IF (EipIntInput[7]=1 AND nOldEipInput[7]<>1) OR exeStop_os THEN
	exeStop_os := FALSE;
	exeStop := NOT exeStop;
	EipIntOutput[8] := 1 - EipIntOutput[8];
END_IF
nOldEipInput[7] := EipIntInput[7];

IF EipIntInput[8]=1 OR exeresetPB THEN
	exeresetPB := FALSE;
	exereset := TRUE;
//ELSE
//	exereset := FALSE;
END_IF

IF EipIntInput[9]=1 OR exerestartPB THEN
	exerestart := TRUE;
ELSE
	exerestart := FALSE;
END_IF

FOR i:=1 TO 2 DO
	IF bMoverEnable[i]= TRUE THEN
		EipIntOutput[i] :=1;
	ELSE
		EipIntOutput[i] :=0;
	END_IF
	IF bMoverDisable[i]= TRUE THEN
		EipIntOutput[i+2] :=1;
	ELSE
		EipIntOutput[i+2] :=0;
	END_IF
END_FOR

//速度変数を外部PLCから変更
IF EipIntInput[10] <> nOldEipInput[10] THEN
	ValueV := EipIntInput[10];
	nOldEipInput[10] := EipIntInput[10];
END_IF
EipIntOutput[6] := ValueV;
IF EipIntInput[11] <> nOldEipInput[11] THEN
	ValueC := EipIntInput[11];
	nOldEipInput[11] := EipIntInput[11];
END_IF
EipIntOutput[7] := ValueC;

IF fbAutoScan.bDone THEN
	EipIntOutput[9] := 1;
ELSE
	EipIntOutput[9] := 0;
END_IF
END_ACTION

END_PROGRAM

// ---- POUs/FB/FB_XpEnableMover.TcPOU
FUNCTION_BLOCK FB_XpEnableMover
VAR_IN_OUT
	XpMover							: MC_PlanarMover;
	XpGroup							: MC_PlanarGroup;
END_VAR
VAR_INPUT
	execute							: BOOL;
END_VAR
VAR_OUTPUT
	done							: BOOL;
	busy							: BOOL;
	error							: BOOL;
	aborted							: BOOL;
END_VAR
VAR
	_XpFeedback						: ARRAY [0.._MAX_XPLANAR_FEEDBACK] OF MC_PlanarFeedback;
END_VAR
VAR
	_sequence						: UINT;
	_i								: UINT;
	_countError						: UINT;
END_VAR
VAR CONSTANT
	_MAX_XPLANAR_FEEDBACK			: UINT := 1;
	_MAX_COUNT_ERROR				: UINT := 5;
	
	_INIT							: UINT := 0000;
	_READY							: UINT := 0001;
	_ENABLE_MOVER					: UINT := 0011;
	_CHECK_ENABLE_MOVER				: UINT := 0012;
	_ADD_TO_GROUP					: UINT := 0013;
	_CHECK_ADD_TO_GROUP				: UINT := 0014;
	_DONE							: UINT := 1000;
	_ERROR							: UINT := 2000;
	_ABORTED						: UINT := 3000;
END_VAR

updateXPlanarFB();
CASE _sequence OF
	_INIT:
		_sequence := _READY;	

	_READY:
		IF execute THEN
			busy := TRUE;
			_sequence := _ENABLE_MOVER;
		END_IF

	_ENABLE_MOVER:
		XpMover.Enable(commandFeedback:= _XpFeedback[0]);
		_sequence := _CHECK_ENABLE_MOVER;
	
	_CHECK_ENABLE_MOVER:
		IF _XpFeedback[0].Done THEN
			_countError := 0;
			_sequence := _ADD_TO_GROUP;
		ELSIF _XpFeedback[0].Error THEN
			_countError := _countError + 1;
			_sequence := _ENABLE_MOVER;
		END_IF
		IF _countError > _MAX_COUNT_ERROR THEN
			_countError := 0;
			_sequence := _ERROR;
		END_IF
	
	_ADD_TO_GROUP:
		XpMover.AddToGroup(commandFeedback:= _XpFeedback[1], group:= XpGroup);
		_sequence := _CHECK_ADD_TO_GROUP;
	
	_CHECK_ADD_TO_GROUP:
		IF _XpFeedback[1].Done THEN
			_countError := 0;
			_sequence := _DONE;
		ELSIF _XpFeedback[1].Error THEN
			_countError := _countError + 1;
			_sequence := _ADD_TO_GROUP;
		END_IF
		IF _countError > _MAX_COUNT_ERROR THEN
			_countError := 0;
			_sequence := _ERROR;
		END_IF
	
	_DONE:
		done := TRUE;
		busy := FALSE;
		IF NOT execute THEN
			done := FALSE;
			_sequence := _READY;
		END_IF
		
	_ERROR:
		error := TRUE;
		busy := FALSE;
		IF NOT execute THEN
			error := FALSE;
			_sequence := _READY;
		END_IF
		
	_ABORTED:
		aborted := TRUE;
		busy := FALSE;
		IF NOT execute THEN
			aborted := FALSE;
			_sequence := _READY;
		END_IF
END_CASE

ACTION updateXPlanarFB:
FOR _i:=0 TO _MAX_XPLANAR_FEEDBACK DO
	_XpFeedback[_i].Update();
END_FOR
END_ACTION

END_FUNCTION_BLOCK

// ---- POUs/FB/FB_XpDisableMover.TcPOU
FUNCTION_BLOCK FB_XpDisableMover
VAR_IN_OUT
	XpMover							: MC_PlanarMover;
	XpGroup							: MC_PlanarGroup;
END_VAR
VAR_INPUT
	execute							: BOOL;
END_VAR
VAR_OUTPUT
	done							: BOOL;
	busy							: BOOL;
	error							: BOOL;
	aborted							: BOOL;
END_VAR
VAR
	_XpFeedback						: ARRAY [0.._MAX_XPLANAR_FEEDBACK] OF MC_PlanarFeedback;
END_VAR
VAR
	_sequence						: UINT;
	_i								: UINT;
	_countError						: UINT;
END_VAR
VAR CONSTANT
	_MAX_XPLANAR_FEEDBACK			: UINT := 1;
	_MAX_COUNT_ERROR				: UINT := 5;
	
	_INIT							: UINT := 0000;
	_READY							: UINT := 0001;
	_REMOVE_FROM_GROUP				: UINT := 0011;
	_CHECK_REMOVE_FROM_GROUP		: UINT := 0012;
	_DISABLE_MOVER					: UINT := 0013;
	_CHECK_DISABLE_MOVER			: UINT := 0014;
	_DONE							: UINT := 1000;
	_ERROR							: UINT := 2000;
	_ABORTED						: UINT := 3000;
END_VAR

updateXPlanarFB();
CASE _sequence OF
	_INIT:
		_sequence := _READY;
		
	_READY:
		IF execute THEN
			busy := TRUE;
			_sequence := _REMOVE_FROM_GROUP;
		END_IF

	_REMOVE_FROM_GROUP:
		XpMover.RemoveFromGroup(commandFeedback:= _XpFeedback[0]);
		_sequence := _CHECK_REMOVE_FROM_GROUP;
	
	_CHECK_REMOVE_FROM_GROUP:
		IF _XpFeedback[0].Done THEN
			_countError := 0;
			_sequence := _DISABLE_MOVER;
		ELSIF _XpFeedback[0].Error THEN
			_countError := _countError + 1;
			_sequence := _REMOVE_FROM_GROUP;
		END_IF
		IF _countError > _MAX_COUNT_ERROR THEN
			_countError := 0;
			_sequence := _ERROR;
		END_IF
	
	_DISABLE_MOVER:
		XpMover.Disable(commandFeedback:= _XpFeedback[1]);
		_sequence := _CHECK_DISABLE_MOVER;
	
	_CHECK_DISABLE_MOVER:
		IF _XpFeedback[1].Done THEN
			_countError := 0;
			_sequence := _DONE;
		ELSIF _XpFeedback[1].Error THEN
			_countError := _countError + 1;
			_sequence := _DISABLE_MOVER;
		END_IF
		IF _countError > _MAX_COUNT_ERROR THEN
			_countError := 0;
			_sequence := _ERROR;
		END_IF
	
	_DONE:
		done := TRUE;
		busy := FALSE;
		IF NOT execute THEN
			done := FALSE;
			_sequence := _READY;
		END_IF
		
	_ERROR:
		error := TRUE;
		busy := FALSE;
		IF NOT execute THEN
			error := FALSE;
			_sequence := _READY;
		END_IF
		
	_ABORTED:
		aborted := TRUE;
		busy := FALSE;
		IF NOT execute THEN
			aborted := FALSE;
			_sequence := _READY;
		END_IF
END_CASE

ACTION updateXPlanarFB:
FOR _i:=0 TO _MAX_XPLANAR_FEEDBACK DO
	_XpFeedback[_i].Update();
END_FOR
END_ACTION

END_FUNCTION_BLOCK

// ---- POUs/FB/FB_XpEnableGroup.TcPOU
FUNCTION_BLOCK FB_XpEnableGroup
VAR_IN_OUT
	XpGroup							: MC_PlanarGroup;
END_VAR
VAR_INPUT
	execute							: BOOL;
END_VAR
VAR_OUTPUT
	done							: BOOL;
	busy							: BOOL;
	error							: BOOL;
	aborted							: BOOL;
END_VAR
VAR
	_XpFeedback						: ARRAY [0.._MAX_XPLANAR_FEEDBACK] OF MC_PlanarFeedback;
END_VAR
VAR
	_sequence						: UINT;
	_i								: UINT;
	_countError						: UINT;
END_VAR
VAR CONSTANT
	_MAX_XPLANAR_FEEDBACK			: UINT := 1;
	_MAX_COUNT_ERROR				: UINT := 5;
	
	_INIT							: UINT := 0000;
	_READY							: UINT := 0001;
	_ENABLE_GROUP					: UINT := 0011;
	_CHECK_ENABLE_GROUP				: UINT := 0012;
	_DONE							: UINT := 1000;
	_ERROR							: UINT := 2000;
	_ABORTED						: UINT := 3000;
END_VAR

updateXPlanarFB();
CASE _sequence OF
	_INIT:
		_sequence := _READY;
		
	_READY:
		IF execute THEN
			busy := TRUE;
			_sequence := _ENABLE_GROUP;
		END_IF

	_ENABLE_GROUP:
		XpGroup.Enable(commandFeedback:= _XpFeedback[0]);
		_sequence := _CHECK_ENABLE_GROUP;
	
	_CHECK_ENABLE_GROUP:
		IF _XpFeedback[0].Done THEN
			_countError := 0;
			_sequence := _DONE;
		ELSIF _XpFeedback[0].Error THEN
			_countError := _countError + 1;
			_sequence := _ENABLE_GROUP;
		END_IF
		IF _countError > _MAX_COUNT_ERROR THEN
			_countError := 0;
			_sequence := _ERROR;
		END_IF
	_DONE:
		done := TRUE;
		busy := FALSE;
		IF NOT execute THEN
			done := FALSE;
			_sequence := _READY;
		END_IF
		
	_ERROR:
		error := TRUE;
		busy := FALSE;
		IF NOT execute THEN
			error := FALSE;
			_sequence := _READY;
		END_IF
		
	_ABORTED:
		aborted := TRUE;
		busy := FALSE;
		IF NOT execute THEN
			aborted := FALSE;
			_sequence := _READY;
		END_IF
END_CASE

ACTION updateXPlanarFB:
FOR _i:=0 TO _MAX_XPLANAR_FEEDBACK DO
	_XpFeedback[_i].Update();
END_FOR
END_ACTION

END_FUNCTION_BLOCK

// ---- POUs/FB/FB_XpEnableEnvironment.TcPOU
FUNCTION_BLOCK FB_XpEnableEnvironment
VAR_IN_OUT
	XpEnvironment					: MC_PlanarEnvironment;
	XpGroup							: MC_PlanarGroup;
END_VAR
VAR_INPUT
	execute							: BOOL;
END_VAR
VAR_OUTPUT
	done							: BOOL;
	busy							: BOOL;
	error							: BOOL;
	aborted							: BOOL;
END_VAR
VAR
	_XpFeedback						: ARRAY [0.._MAX_XPLANAR_FEEDBACK] OF MC_PlanarFeedback;
END_VAR
VAR
	_sequence						: UINT;
	_i								: UINT;
	_countError						: UINT;
END_VAR
VAR CONSTANT
	_MAX_XPLANAR_FEEDBACK			: UINT := 1;
	_MAX_COUNT_ERROR				: UINT := 5;
	
	_INIT							: UINT := 0000;
	_READY							: UINT := 0001;
	_CREATE_BOUNDARY				: UINT := 0011;
	_CHECK_CREATE_BOUNDARY			: UINT := 0012;
	_ENVIRONMENT_ADD_TO_GROUP		: UINT := 0013;
	_CHECK_ENVIRONMENT_ADD_TO_GROUP	: UINT := 0014;
	_DONE							: UINT := 1000;
	_ERROR							: UINT := 2000;
	_ABORTED						: UINT := 3000;
END_VAR

updateXPlanarFB();
CASE _sequence OF
	_INIT:
		_sequence := _READY;
		
	_READY:
		IF execute THEN
			busy := TRUE;
			_sequence := _CREATE_BOUNDARY;
		END_IF
		
	_CREATE_BOUNDARY:
		XpEnvironment.CreateBoundary(commandFeedback:= _XpFeedback[0]);
		_sequence := _CHECK_CREATE_BOUNDARY;
	
	_CHECK_CREATE_BOUNDARY:
		IF _XpFeedback[0].Done THEN
			_countError := 0;
			_sequence := _ENVIRONMENT_ADD_TO_GROUP;
		ELSIF _XpFeedback[0].Error THEN
			_countError := _countError + 1;
			_sequence := _CREATE_BOUNDARY;
		END_IF
		IF _countError > _MAX_COUNT_ERROR THEN
			_countError := 0;
			_sequence := _ERROR;
		END_IF
	
	_ENVIRONMENT_ADD_TO_GROUP:
		XpEnvironment.AddToGroup(commandFeedback:= _XpFeedback[1], group:= XpGroup);
		_sequence := _CHECK_ENVIRONMENT_ADD_TO_GROUP;
	
	_CHECK_ENVIRONMENT_ADD_TO_GROUP:
		IF _XpFeedback[1].Done THEN
			_countError := 0;
			_sequence := _DONE;
		ELSIF _XpFeedback[1].Error THEN
			_countError := _countError + 1;
			_sequence := _ENVIRONMENT_ADD_TO_GROUP;
		END_IF
		IF _countError > _MAX_COUNT_ERROR THEN
			_countError := 0;
			_sequence := _ERROR;
		END_IF
		
	_DONE:
		done := TRUE;
		busy := FALSE;
		IF NOT execute THEN
			done := FALSE;
			_sequence := _READY;
		END_IF
		
	_ERROR:
		error := TRUE;
		busy := FALSE;
		IF NOT execute THEN
			error := FALSE;
			_sequence := _READY;
		END_IF
		
	_ABORTED:
		aborted := TRUE;
		busy := FALSE;
		IF NOT execute THEN
			aborted := FALSE;
			_sequence := _READY;
		END_IF
END_CASE

ACTION updateXPlanarFB:
FOR _i:=0 TO _MAX_XPLANAR_FEEDBACK DO
	_XpFeedback[_i].Update();
END_FOR
END_ACTION

END_FUNCTION_BLOCK

// ---- POUs/FB/FB_XpEnableTrack.TcPOU
FUNCTION_BLOCK FB_XpEnableTrack
VAR_IN_OUT
	xpTrack							: MC_PlanarTrack;
	xpGroup							: MC_PlanarGroup;
END_VAR
VAR_INPUT
	execute							: BOOL;
END_VAR
VAR_OUTPUT
	done							: BOOL;
	busy							: BOOL;
	error							: BOOL;
	aborted							: BOOL;
END_VAR
VAR
	_XpFeedback						: ARRAY [0.._MAX_XPLANAR_FEEDBACK] OF MC_PlanarFeedback;
END_VAR
VAR
	_sequence						: UINT;
	_i								: UINT;
	_countError						: UINT;
END_VAR
VAR CONSTANT
	_MAX_XPLANAR_FEEDBACK			: UINT := 1;
	_MAX_COUNT_ERROR				: UINT := 5;
	
	_INIT							: UINT := 0000;
	_READY							: UINT := 0001;
	_ENABLE_TRACK					: UINT := 0011;
	_CHECK_ENABLE_TRACK				: UINT := 0012;
	_TRACK_ADD_TO_GROUP				: UINT := 0013;
	_CHECK_TRACK_ADD_TO_GTOUP		: UINT := 0014;
	_DONE							: UINT := 1000;
	_ERROR							: UINT := 2000;
	_ABORTED						: UINT := 3000;
END_VAR

updateXPlanarFB();
CASE _sequence OF
	_INIT:
		_sequence := _READY;

	_READY:
		IF execute THEN
			busy := TRUE;
			_sequence := _ENABLE_TRACK;
		END_IF

	_ENABLE_TRACK:
		xpTrack.Enable(commandFeedback:= _xpFeedback[0]);
		_sequence := _CHECK_ENABLE_TRACK;
		
	_CHECK_ENABLE_TRACK:
		IF _XpFeedback[0].Done THEN
			_countError := 0;
			_sequence := _TRACK_ADD_TO_GROUP;
		ELSIF _XpFeedback[0].Error THEN
			_countError := _countError + 1;
			_sequence := _ENABLE_TRACK;
		END_IF
		IF _countError > _MAX_COUNT_ERROR THEN
			_countError := 0;
			_sequence := _ERROR;
		END_IF
		
	_TRACK_ADD_TO_GROUP:
		xpTrack.AddToGroup(commandFeedback:= _xpFeedback[1], group:= xpGroup);
		_sequence := _CHECK_TRACK_ADD_TO_GTOUP;
	
	_CHECK_TRACK_ADD_TO_GTOUP:
		IF _XpFeedback[1].Done THEN
			_countError := 0;
			_sequence := _DONE;
		ELSIF _XpFeedback[1].Error THEN
			_countError := _countError + 1;
			_sequence := _TRACK_ADD_TO_GROUP;
		END_IF
		IF _countError > _MAX_COUNT_ERROR THEN
			_countError := 0;
			_sequence := _ERROR;
		END_IF
		
	_DONE:
		done := TRUE;
		busy := FALSE;
		IF NOT execute THEN
			done := FALSE;
			_sequence := _READY;
		END_IF
		
	_ERROR:
		error := TRUE;
		busy := FALSE;
		IF NOT execute THEN
			error := FALSE;
			_sequence := _READY;
		END_IF
		
	_ABORTED:
		aborted := TRUE;
		busy := FALSE;
		IF NOT execute THEN
			aborted := FALSE;
			_sequence := _READY;
		END_IF
END_CASE

ACTION updateXPlanarFB:
FOR _i:=0 TO _MAX_XPLANAR_FEEDBACK DO
	_xpFeedback[_i].Update();
END_FOR
END_ACTION

END_FUNCTION_BLOCK

// ---- POUs/FB/FB_XPlanarAutoScan.TcPOU
FUNCTION_BLOCK FB_XPlanarAutoScan
VAR_INPUT
    bExecute    : BOOL; 
END_VAR
VAR_OUTPUT
    bBusy       : BOOL;
    bDone       : BOOL;
    bError      : BOOL;
END_VAR
VAR
    nState      : INT := 0;
    rtExecute   : R_TRIG;
    
    fbEnv       : FB_TcIoXPlanarEnvironment;
    ipXpu       : I_TcIoXPlanarProcessingUnit;
END_VAR

rtExecute(CLK := bExecute);

IF rtExecute.Q THEN
    bBusy  := TRUE;
    bDone  := FALSE;
    bError := FALSE;
    nState := 10; 
END_IF

CASE nState OF
    0: //wait

    10: 
        IF fbEnv.Init(bExecute := TRUE) THEN
            nState := 20;
        END_IF

    20: 
        ipXpu := fbEnv.TcIoXpu(nNum := 1); 
        
        IF ipXpu <> 0 THEN
            nState := 30;
        ELSE
            bError := TRUE;
            bBusy  := FALSE;
            nState := 0;
        END_IF

    30: 
        IF ipXpu.SetCoordMoverCommunicationCmd(	
			CoordinatedMoverCommCommand.IdentifyAndAssignPossible) THEN
            bBusy  := FALSE;
            bDone  := TRUE;
            nState := 0;
        END_IF
        
END_CASE

END_FUNCTION_BLOCK

// ---- POUs/FB/FB_XpMoverState.TcPOU

{attribute 'no_assign'}
FUNCTION_BLOCK FB_XpMoverState
VAR_INPUT
	eTaskMover 			: E_Movertask :=1;
//	refMover			: REFERENCE TO MC_PlanarMover;
	bResetMover			: BOOL;
	bRestartMover		: BOOL;
	nMoverState			: INT :=0 ;
	TargetNo			: INT;
	bNextStep			: BOOL;
END_VAR
VAR_OUTPUT
	bDoneMover 		:BOOL;
END_VAR
VAR_IN_OUT
	stParams : ST_MoverParams;
	refMover 	: MC_PlanarMover;
	refTrack	: ARRAY [1..gvl.MAX_TRACK] OF MC_PlanarTrack;
	reftrail	: MC_PlanarTrackTrail;
END_VAR
VAR
	MSFeedback			: ARRAY [0..30] OF MC_PlanarFeedback;
	GrFeedback			: ARRAY [0..30] OF MC_PlanarFeedbackGearInPosOnTrackWithMasterMover;
	
//	bDoneMover			: BOOL;
	//eTaskMover			: E_MOVERTASK;
	
	stOption			: ARRAY [1..2] OF ST_MoveOnTrackOptions;
	Constraint			: ARRAY [1..2] OF DynamicConstraint_PathXY;
	Constraint_c		: DynamicConstraint_Coordinates;
	stoption_c			: ST_MoveCOptions;
	stOption_j			: ST_JoinTrackOptions;
	stOption_l			: ST_LeaveTrackOptions;
	i: INT;
	ValueC				: LREAL := 300;
	stTargetPos			: LREAL;
	LeavePosition		: ARRAY [2..3] OF PositionXYC;

	fMasterSyncDist: INT;
	fSlaveSyncDist: INT;
END_VAR

IF ADR(refMover) = 0 THEN
	RETURN;
END_IF

IF bRestartMover THEN
	bRestartMover := FALSE;
	nMoverState := 0;
	eTaskMover := E_MoverTask.IDLE;
	bNextStep := FALSE;
	RETURN;
END_IF

IF bResetMover THEN
	bResetMover := FALSE;
	nMoverState := 950;
	eTaskMover := E_MoverTask.RESET_ERROR;
	bNextStep := FALSE;
END_IF

CASE nMoverState OF
	0://IDLE
	IF eTaskMover =E_MoverTask.IDLE THEN //IDLE状態で0に戻ったらbDoneMoverを0に戻す
	bDoneMover := FALSE;
	END_IF
	
		CASE eTaskMover OF
			E_MoverTask.JOIN				: nMoverState :=100;
			E_MoverTask.MOVE_TRACK			: nMoverState :=200;
			E_MoverTask.MOVE_C_ROTATE		: nMoverState :=300;
			E_MoverTask.RESET_ROTATE		: nMoverState :=900;
			E_Movertask.RESET_ERROR			: nMoverState :=950;
		END_CASE
	
	100://JOIN
	refMover.JoinTrack(commandFeedback:= MSFeedback[1], 
				targetTrack:= refTrack[TargetNo], //TargetNo = TrackNo
				constraint:= constraint[2], 
				options:= stOption_j);
	nMoverState:=101;
	
	101:
	IF (MSFeedback[1].Active OR MSFeedback[1].Done) THEN
		nMoverState:=102;
	END_IF	
	
	102:
	IF MSFeedback[1].Done THEN
		bDoneMover := TRUE;
		nMoverState := 0;
	END_IF

	
	200://MOVE Track
	refMover.MoveOnTrack(
		commandFeedback:= MSFeedback[2], 
		targetTrack:= refTrack[1], 
		targetPositionOnTrack:= refTrack[TargetNo].GetLength(),
		constraint:= Constraint[1], 
		options:= stOption[1]);
		nMoverState:=201;
	
	201:
	IF (MSFeedback[2].Active OR MSFeedback[2].Done OR bNextStep) THEN
		nMoverState:=202;
	END_IF	
	
	202:
	IF MSFeedback[2].Done OR bNextStep THEN
		bDoneMover := TRUE;
		nMoverState := 0;
	END_IF
	
	300:
	//足し算
	stTargetPos := refMover.MCTOPLC.SET.SetPos.c + 720;
	//C回転
	refMover.MoveC(commandFeedback:=MSFeedback[3] ,
			targetPosition:=stTargetPos ,
			constraint:=constraint_c ,
			options:=stOption_c);
	nMoverState :=301;
	
	301:
	IF (MSFeedback[3].Active OR MSFeedback[3].Done) THEN
		nMoverState:=302;
	END_IF	
	
	302:
	IF MSFeedback[3].Done THEN
		bDoneMover := TRUE;
		nMoverState := 0;
	END_IF	
	
	(*
	900:
	IF NOT refMover.MCTOPLC.STD.Busy THEN
		refMover.SetPosition(commandFeedback := MSFeedback[29],
			position := [refMover.MCTOPLC.ACT.ActPos.x,
						refMover.MCTOPLC.ACT.ActPos.y,
						refMover.MCTOPLC.ACT.ActPos.z,
						refMover.MCTOPLC.ACT.ActPos.a,
						refMover.MCTOPLC.ACT.ActPos.b,
						0]);
	END_IF
	*)
	950:
	refMover.Reset(commandFeedBack :=MSFeedback[30]);
	nMoverState :=951;
	
	951:
	IF MSFeedback[30].Active OR MSFeedback[30].Done THEN
		nMoverState :=952;
	END_IF
	
	952:
	IF MSFeedback[30].Done THEN
		bDoneMover :=TRUE;
		nMoverState := 0;
	END_IF
		
END_CASE


stOption[1].gap := 170.0;
stOption[2].gap := 170.0 (*118.0*);

constraint[1].SetValuesVADJ(
			V:= 150,
			A:= 7000,
			D:= 7000,
			J:= 3000);

Constraint[2].SetValuesVADJ(
		V:= stParams.lrVelocity, 
		A:= 7000, 
		D:= 7000,
		J:=35000);
		
Constraint_c.SetLimit(
	Coordinate:= Coord_Mcs_C1, 
	V:= stParams.lrVelocity_c, 
	A:= 7000, 
	D:= 7000, 
	J:= 35000);
	


(*
refMover.Update();
*)
FOR i:=0 TO 30 DO
	MSFeedback[i].Update();
	GrFeedback[i].Update();
END_FOR

END_FUNCTION_BLOCK

// ---- POUs/FB/FB_XpMoverInit.TcPOU
FUNCTION_BLOCK FB_XpMoverInit
VAR_INPUT
	exeXpEnableMover_Ind 	: BOOL;
	exeXpDisableMover_Ind 	: BOOL;
	exereset : BOOL;
END_VAR
VAR_OUTPUT
END_VAR
VAR_IN_OUT
	refMover 	: MC_PlanarMover;
	xpGroup		: MC_planargroup;
END_VAR
VAR
	nState : E_State :=0;
	MSFeedback				: ARRAY [0..30] OF MC_PlanarFeedback;
	constraint				: DynamicConstraint_PathXY;
	i: INT;
	ErrorID : LREAL;
	fbTimer: TON;
	stTargetPos	: PositionXYC ;

END_VAR

IF exeXpEnableMover_Ind AND refMover.MCTOPLC.STD.State = MC.MC_PLANAR_STATE.Disabled THEN //運転準備ボタン押下かつステート0のとき
	nState := E_State.EnableMover;
	exeXpEnableMover_Ind := FALSE;
END_IF

IF exeXpDisableMover_Ind AND refMover.MCTOPLC.STD.State = MC.MC_PLANAR_STATE.Enabled THEN//運転終了ボタン押下かつステート30のとき
	nState := E_State.DisableMover;
	exeXpDisableMover_Ind := FALSE;
END_IF

IF refMover.Error THEN
	ErrorID := refMover.ErrorId;
	nState:=E_State.ERROR;
END_IF

CASE nState OF
	E_State.init:
	refMover.Reset(commandFeedback:=MSFeedback[0]);
	nState :=E_State.INIT2;
	
	E_State.INIT2:
	IF MSFeedback[0].Done THEN
		fbTimer(IN:= TRUE, PT:=T#200MS);
		IF fbTimer.Q THEN
			fbTimer(IN := FALSE);
		END_IF	
	END_IF
	
	
	E_State.EnableMover://moverを有効化（浮上）
		refMover.Enable(commandFeedback:= MSFeedback[10]);
		nState :=E_State.EnableCheck;
		//nState :=E_State.AddToGroup;
	
	E_State.EnableCheck://mover状態確認
	IF MSFeedback[10].Error THEN
		nState :=E_State.ERROR;//エラー状態のためno.999	に遷移
	ELSIF MSFeedback[10].Done THEN
		stTargetPos.x := refMover.MCTOPLC.ACT.ActPos.x;
		stTargetPos.y := refMover.MCTOPLC.ACT.ActPos.y;
		stTargetPos.c := refMover.MCTOPLC.ACT.ActPos.c;
		refMover.MoveToPosition(commandFeedback:=MSFeedback[1],
					targetPosition:=stTargetPos,
					constraint :=constraint,
					options := 0);
		nState :=E_State.PositionCheck;//すべてdoneのため次のステートに進む
	END_IF
	
	E_State.PositionCheck:
	IF MSFeedback[1].Done THEN
		nState := e_state.AddToGroup;
	END_IF
	
	E_State.AddToGroup://moverとtrackをxpgroupに追加
	IF refMover.MCTOPLC.STD.GroupOID <> 0 THEN
		nState := e_state.AddToGroupCheck;
	ELSE
		refMover.AddToGroup(commandfeedback := MSFeedback[12],group:= XpGroup);
		nState := E_State.AddToGroupCheck;
	END_IF
	refMover.AddToGroup(commandfeedback := MSFeedback[12],group:= XpGroup);
	nState := E_State.AddToGroupCheck;
	
	E_State.AddToGroupCheck:
	IF MSFeedback[12].Error THEN
		nState :=E_State.ERROR;
	ELSIF MSFeedback[12].Done THEN
		nState := E_State.EnableComp;
	END_IF
	
	E_State.EnableComp://Enable完了表示
	//stay

	E_State.DisableMover://moverを無効化（下ろす）
	refMover.Disable(commandFeedback := MSFeedback[13]);
	nState := E_State.DisableCheck;
	
	E_State.DisableCheck://mover状態確認
	IF MSFeedback[13].Error THEN
		nState :=E_State.ERROR;
	ELSIF MSFeedback[13].Done THEN
		nState := E_State.DisableComp;
	END_IF
	
	E_State.DisableComp:	//Disable完了表示
	nState := E_State.INIT;
	
	E_State.ERROR:
	IF exereset THEN;
		exereset :=FALSE;
		nState :=E_State.INIT;
	END_IF
END_CASE

FOR i := 0 TO 30 DO
	MSFeedback[i].Update();
END_FOR
	
	Constraint.SetValuesVADJ(
		V:= 500, 
		A:= 7000, 
		D:= 7000,
		J:=35000);

END_FUNCTION_BLOCK

// ---- POUs/FB/FB_XpMoverPara.TcPOU
FUNCTION_BLOCK FB_XpMoverPara
VAR_IN_OUT
	bBeforeLink		: BOOL;
	bT2Busy			: BOOL;
	fbMoverSeq		: FB_XpMoverState;
END_VAR
VAR_INPUT
	bJoinDone		: BOOL;
	bT2Available	: BOOL;
	bT3Available	: BOOL;
	exestop			: BOOL;
END_VAR
VAR_OUTPUT
	eTaskMover		: E_MoverTask;
END_VAR
VAR
	nGearingState	: INT;
END_VAR

	CASE nGearingState OF
		0:
		IF bJoinDone THEN
			nGearingState :=50;
		END_IF
		
		50://Move To T1
		IF NOT exestop THEN
			fbMoverSeq.TargetNo := 1;
			fbMoverSeq.eTaskMover := E_MoverTask.MOVE_TRACK;
			nGearingState := 51;
		END_IF
		
		51:
		IF fbMoverSeq.bDoneMover THEN
			fbMoverSeq.eTaskMover :=E_MoverTask.IDLE;
			nGearingState :=100;
		END_IF
		
		100://Track select T2 or T3
		IF bT2Available AND NOT bT2Busy THEN
			fbMoverSeq.TargetNo := 5; //track2
			bT2Busy :=TRUE;
		ELSIF bT3Available THEN
			fbMoverSeq.TargetNo := 4; //track3
		END_IF
		nGearingState :=101;
		
		101:
		fbMoverSeq.eTaskMover := E_MoverTask.MOVE_TRACK;
		nGearingState := 110;

		110:
		IF fbMoverSeq.bDoneMover THEN
			fbMoverSeq.eTaskMover := E_MoverTask.IDLE;
			IF fbMoverSeq.TargetNo = 5 THEN
				nGearingState :=120;
			ELSIF fbMoverSeq.TargetNo = 4 THEN
				bBeforeLink := TRUE;
				nGearingState :=121;
			END_IF
		END_IF
		
		120://T2 Mastar
		IF bBeforeLink THEN
			fbMoverSeq.TargetNo := 2;
			nGearingState := 130;
		END_IF
		
		121:
		fbMoverSeq.TargetNo := 3;
		nGearingState :=131;
		
		130:	
		fbMoverSeq.eTaskMover := E_MoverTask.MOVE_TRACK;
		nGearingState := 140;
	
		140:
		IF fbMoverSeq.bDoneMover THEN
			fbMoverSeq.eTaskMover :=E_MoverTask.IDLE;
			IF fbMoverSeq.TargetNo = 2 THEN
				bT2Busy := FALSE;
			ELSIF fbMoverSeq.TargetNo = 3 THEN
				bBeforeLink := FALSE;
			END_IF
			nGearingState :=300;
		END_IF

		300:
		IF NOT exeStop THEN
			nGearingState := 50;
		END_IF
		
	END_CASE

END_FUNCTION_BLOCK

// ---- POUs/FB/FB_XpJoinTrack.TcPOU
FUNCTION_BLOCK FB_XpJoinTrack
VAR_IN_OUT
	XpMover							: MC_PlanarMover;
	XpTrack							: MC_PlanarTrack;
END_VAR
VAR_INPUT
	execute							: BOOL;
	velocity						: LREAL := 100;
	acceleration					: LREAL := 2000;
	jerk							: LREAL := 20000;
END_VAR
VAR_OUTPUT
	done							: BOOL;
	busy							: BOOL;
	error							: BOOL;
	aborted							: BOOL;
END_VAR
VAR
	_XpFeedback						: ARRAY [0.._MAX_XPLANAR_FEEDBACK] OF MC_PlanarFeedback;
	_XpCondition		 			: DynamicConstraint_PathXY;
END_VAR
VAR
	_sequence						: UINT;
	_i								: UINT;
	_countError						: UINT;
	_velocity						: LREAL;
	_acceleration					: LREAL;
	_jerk							: LREAL;
END_VAR
VAR CONSTANT
	_MAX_XPLANAR_FEEDBACK			: UINT := 1;
	_MAX_COUNT_ERROR				: UINT := 5;
	
	_INIT							: UINT := 0000;
	_READY							: UINT := 0001;
	_JOIN_TRACK						: UINT := 0011;
	_CHECK_JOIN_TRACK				: UINT := 0012;
	_DONE							: UINT := 1000;
	_ERROR							: UINT := 2000;
	_ABORTED						: UINT := 3000;
END_VAR

updateXPlanarFB();
CASE _sequence OF
	_INIT:
		_sequence := _READY;
		
	_READY:
		IF execute THEN
			busy := TRUE;
			_sequence := _JOIN_TRACK;
			setInputVariables();
		END_IF
		
	_JOIN_TRACK:
		_XpCondition.SetValuesVADJ(
			V:= _velocity, 
			A:= _acceleration, 
			D:= _acceleration, 
			J:= _jerk);
		XpMover.JoinTrack(commandFeedback:= _XpFeedback[0], 
			targetTrack:= XpTrack, 
			constraint:= _XpCondition, 
			options:= 0);
		_sequence := _CHECK_JOIN_TRACK;
		
	_CHECK_JOIN_TRACK:
		IF _XpFeedback[0].Done THEN
			_countError := 0;
			_sequence := _DONE;
		ELSIF _XpFeedback[0].Error THEN
			_countError := _countError + 1;
			_sequence := _JOIN_TRACK;
		ELSIF _XpFeedback[0].Aborted THEN
			_countError := 0;
			_sequence := _ABORTED;
		END_IF
		IF _countError > _MAX_COUNT_ERROR THEN
			_countError := 0;
			_sequence := _ERROR;
		END_IF
		
	_DONE:
		done := TRUE;
		busy := FALSE;
		IF NOT execute THEN
			done := FALSE;
			_sequence := _READY;
		END_IF
	
	_ERROR:
		error := TRUE;
		busy := FALSE;
		IF NOT execute THEN
			error := FALSE;
			_sequence := _READY;
		END_IF
		
	_ABORTED:
		aborted := TRUE;
		busy := FALSE;
		IF NOT execute THEN
			aborted := FALSE;
			_sequence := _READY;
		END_IF
END_CASE

ACTION setInputVariables:
_velocity := velocity;
_acceleration := acceleration;
_jerk := jerk;
END_ACTION

ACTION updateXPlanarFB:
FOR _i:=0 TO _MAX_XPLANAR_FEEDBACK DO
	_XpFeedback[_i].Update();
END_FOR
END_ACTION

END_FUNCTION_BLOCK

// ---- POUs/FB/FB_XpMoveTrack.TcPOU
FUNCTION_BLOCK FB_XpMoveTrack
VAR_IN_OUT
	XpMover							: MC_PlanarMover;
	XpTrack							: MC_PlanarTrack;
END_VAR
VAR_INPUT
	execute							: BOOL;
	distance						: LREAL := 160;
	velocity						: LREAL := 100;
	acceleration					: LREAL := 2000;
	jerk							: LREAL := 20000;
	gap								: LREAL := 170;
	gapmode							: MC_GAP_MODE_ON_TRACK := MC_GAP_MODE_ON_TRACK.Standard1D;
END_VAR
VAR_OUTPUT
	done							: BOOL;
	busy							: BOOL;
	error							: BOOL;
	aborted							: BOOL;
END_VAR
VAR
	_XpFeedback						: ARRAY [0.._MAX_XPLANAR_FEEDBACK] OF MC_PlanarFeedback;
	_XpCondition		 			: DynamicConstraint_PathXY;
	_XpOptionMoveOnTrack			: ST_MoveOnTrackOptions;
END_VAR
VAR
	_sequence						: UINT;
	_i								: UINT;
	_countError						: UINT;
	_distance						: LREAL;
	_velocity						: LREAL;
	_acceleration					: LREAL;
	_jerk							: LREAL;
	_gap							: LREAL;
	_gapmode						: MC_GAP_MODE_ON_TRACK;
END_VAR
VAR CONSTANT
	_MAX_XPLANAR_FEEDBACK			: UINT := 1;
	_MAX_COUNT_ERROR				: UINT := 5;
	
	_INIT							: UINT := 0000;
	_READY							: UINT := 0001;
	_MOVE_ON_TRACK					: UINT := 0011;
	_CHECK_MOVE_ON_TRACK			: UINT := 0012;
	_DONE							: UINT := 1000;
	_ERROR							: UINT := 2000;
	_ABORTED						: UINT := 3000;
END_VAR

updateXPlanarFB();
CASE _sequence OF
	_INIT:
		_sequence := _READY;
		
	_READY:
		IF execute THEN
			busy := TRUE;
			_sequence := _MOVE_ON_TRACK;
			setInputVariables();
		END_IF
		
	_MOVE_ON_TRACK:
		_XpCondition.SetValuesVADJ(
			V:= _velocity, 
			A:= _acceleration, 
			D:= _acceleration, 
			J:= _jerk);
		_XpOptionMoveOnTrack.gap := _gap;
		_XpOptionMoveOnTrack.gapMode := _gapmode;
		XpMover.MoveOnTrack(commandFeedback:= _XpFeedback[0], 
			targetTrack:= XpTrack, 
			//targetPositionOnTrack:= _distance, 
			targetPositionOnTrack:= XpTrack.GetLength(), 
			constraint:= _XpCondition, 
			options:= _XpOptionMoveOnTrack);
		_sequence := _CHECK_MOVE_ON_TRACK;
		
	_CHECK_MOVE_ON_TRACK:
		IF _XpFeedback[0].Done THEN
			_countError := 0;
			_sequence := _DONE;
		ELSIF _XpFeedback[0].Error THEN
			_countError := _countError + 1;
			_sequence := _MOVE_ON_TRACK;
		ELSIF _XpFeedback[0].Aborted THEN
			_countError := 0;
			_sequence := _ABORTED;
		END_IF
		IF _countError > _MAX_COUNT_ERROR THEN
			_countError := 0;
			_sequence := _ERROR;
		END_IF
		
	_DONE:
		done := TRUE;
		busy := FALSE;
		IF NOT execute THEN
			done := FALSE;
			_sequence := _READY;
		END_IF
	
	_ERROR:
		error := TRUE;
		busy := FALSE;
		IF NOT execute THEN
			error := FALSE;
			_sequence := _READY;
		END_IF
		
	_ABORTED:
		aborted := TRUE;
		busy := FALSE;
		IF NOT execute THEN
			aborted := FALSE;
			_sequence := _READY;
		END_IF
END_CASE

ACTION setInputVariables:
_distance := distance;
_velocity := velocity;
_acceleration := acceleration;
_jerk := jerk;
_gap := gap;
_gapmode := gapmode;
END_ACTION

ACTION updateXPlanarFB:
FOR _i:=0 TO _MAX_XPLANAR_FEEDBACK DO
	_XpFeedback[_i].Update();
END_FOR
END_ACTION

END_FUNCTION_BLOCK

// ---- POUs/FB/FB_StationT1.TcPOU
FUNCTION_BLOCK FB_StationT1
VAR_IN_OUT
	XpMover			: MC_PlanarMover;
	XpTrack			: ARRAY[*] OF MC_PlanarTrack;
END_VAR
VAR_INPUT
	execute			: BOOL;
	bT2Ready		: BOOL :=TRUE;
	bT3Ready		: BOOL :=TRUE;
END_VAR
VAR_OUTPUT
	bOccupied		: BOOL;
	bReady			: BOOL;
END_VAR
VAR
	nState			: INT;
	fbMoveTrack		: FB_XpMoveTrack;
	nTargetTrack	: INT;
	bMove			: BOOL;
END_VAR

CASE nState OF
	0://init
	IF execute THEN
		bOccupied := TRUE;//Stationの状態をOccupiedにする
		bReady := FALSE;
		nState := 10;
	END_IF
	
	10://判断
	IF bT2Ready THEN
		nTargetTrack := E_TrackName.T2_1_ToLink;//右ルート
		nState := 20;
	ELSIF bT3Ready THEN
		nTargetTrack := E_TrackName.T3_1_ToLink;//左ルート
		nState := 20;
	END_IF
	
	20://移動
	bMove := TRUE;
	fbMoveTrack(XpMover:= XpMover, 
				XpTrack:= XpTrack[nTargetTrack],
				execute := TRUE);
	IF fbMoveTrack.done THEN
		fbMoveTrack.execute := FALSE;
		bOccupied := FALSE;
		bReady := TRUE;
		bMove := FALSE;
		nState := 40;
	END_IF
	
	40://initへ戻る
	nState := 0;
END_CASE

END_FUNCTION_BLOCK

// ---- POUs/FB/FB_StationT2.TcPOU
FUNCTION_BLOCK FB_StationT2
VAR_IN_OUT
	XpMover			: MC_PlanarMover;
	XpTrack			: ARRAY [*] OF MC_PlanarTrack;
END_VAR
VAR_INPUT
	execute			: BOOL;
	bT3Occupied		: BOOL;
	bT3BeforeRotate	: BOOL;
END_VAR
VAR_OUTPUT
	bOccupied		: BOOL;
	bReady			: BOOL;
END_VAR
VAR
	nState			: INT;
	fbMoveTrack		: FB_XpMoveTrack;
	fbMoveC			: FB_XpMoveC;
	nTargetTrack	: INT;
	bMove			: BOOL;
	bMoveC			: BOOL;
	nRotatePos		: LREAL :=0;
END_VAR

CASE nState OF
	0: //init
	IF execute THEN
		bOccupied := TRUE;//Stationの状態をOccupiedにする
		bReady := FALSE;
		nState := 10;
	END_IF
	
	10://T3のMover待ち
	IF bT3Occupied THEN
		nState := 20;
	END_IF
	
	
	20://移動
	ntargetTrack:= E_TrackName.T2_2_ToRotate;
	fbMoveTrack.execute:= TRUE;
	
	IF fbMoveTrack.done THEN
		fbMoveTrack.execute:= FALSE;
		bOccupied := FALSE;
		bReady := TRUE;//Stationの状態をREADYにする
		nState := 30;
	END_IF
	
	30://回転
	IF bT3BeforeRotate THEN //T3のMoverが到着したら
		fbMoveC.execute:= TRUE;
		IF fbMoveC.done THEN
			fbMoveC.execute := FALSE;
			nState := 40;
		END_IF
	END_IF
	
	40:	//T1へ移動
	nTargetTrack := E_TrackName.T1_1_ToRotate;
	fbMoveTrack.execute:= TRUE;
		nState := 100;
	
	100://initへ
	fbMoveTrack.execute := FALSE;//移動指令を落とす
	nState := 0;
END_CASE

IF bMove THEN
	fbMoveTrack(XpMover:= XpMover, 
				XpTrack:= XpTrack[nTargetTrack]);
ELSIF bMoveC THEN	
	fbMoveC(XpMover:= XpMover, 
			position:= nRotatePos + 360);
END_IF

END_FUNCTION_BLOCK

// ---- POUs/FB/FB_XpMoveC.TcPOU
FUNCTION_BLOCK FB_XpMoveC
VAR_IN_OUT
	XpMover							: MC_PlanarMover;
END_VAR
VAR_INPUT
	execute							: BOOL;
	position						: LREAL := 360;
	velocity						: LREAL := 100;
	acceleration					: LREAL := 2000;
	jerk							: LREAL := 20000;
END_VAR
VAR_OUTPUT
	done							: BOOL;
	busy							: BOOL;
	error							: BOOL;
	aborted							: BOOL;
END_VAR
VAR
	_XpFeedback						: ARRAY [0.._MAX_XPLANAR_FEEDBACK] OF MC_PlanarFeedback;
	_XpCondition		 			: DynamicConstraint_Coordinates;
END_VAR
VAR
	_sequence						: UINT;
	_i								: UINT;
	_countError						: UINT;
	_position						: LREAL;
	_velocity						: LREAL;
	_acceleration					: LREAL;
	_jerk							: LREAL;
END_VAR
VAR CONSTANT
	_MAX_XPLANAR_FEEDBACK			: UINT := 1;
	_MAX_COUNT_ERROR				: UINT := 5;
	
	_INIT							: UINT := 0000;
	_READY							: UINT := 0001;
	_MOVE_C							: UINT := 0011;
	_CHECK_MOVE_C					: UINT := 0012;
	_DONE							: UINT := 1000;
	_ERROR							: UINT := 2000;
	_ABORTED						: UINT := 3000;
END_VAR

updateXPlanarFB();
CASE _sequence OF
	_INIT:
		_XpCondition.AddLimit(
			Coordinate:= Coord_Mcs_C1, 
			V:= velocity, 
			A:= acceleration, 
			D:= acceleration, 
			J:= jerk);
		_sequence := _READY;
	
	_READY:
		IF execute THEN
			busy := TRUE;
			_sequence := _MOVE_C;
			setInputVariables();
		END_IF
		
	_MOVE_C:
		_XpCondition.SetLimit(
			Coordinate:= Coord_Mcs_C1, 
			V:= _velocity, 
			A:= _acceleration, 
			D:= _acceleration, 
			J:= _jerk);
		XpMover.MoveC(commandFeedback:= _XpFeedback[0], 
			targetPosition:= _position, 
			constraint:= _XpCondition, 
			options:= 0);
		_sequence := _CHECK_MOVE_C;
		
	_CHECK_MOVE_C:
		IF _XpFeedback[0].Done THEN
			_countError := 0;
			_sequence := _DONE;
		ELSIF _XpFeedback[0].Error THEN
			_countError := _countError + 1;
			_sequence := _MOVE_C;
		END_IF
		IF _countError > _MAX_COUNT_ERROR THEN
			_countError := 0;
			_sequence := _ERROR;
		END_IF
		
	_DONE:
		done := TRUE;
		busy := FALSE;
		IF NOT execute THEN
			done := FALSE;
			_sequence := _READY;
		END_IF
	
	_ERROR:
		error := TRUE;
		busy := FALSE;
		IF NOT execute THEN
			error := FALSE;
			_sequence := _READY;
		END_IF
		
	_ABORTED:
		aborted := TRUE;
		busy := FALSE;
		IF NOT execute THEN
			aborted := FALSE;
			_sequence := _READY;
		END_IF
END_CASE

ACTION setInputVariables:
_position := position;
_velocity := velocity;
_acceleration := acceleration;
_jerk := jerk;
END_ACTION

ACTION updateXPlanarFB:
FOR _i:=0 TO _MAX_XPLANAR_FEEDBACK DO
	_XpFeedback[_i].Update();
END_FOR
END_ACTION

END_FUNCTION_BLOCK

// ---- POUs/FB/FB_StationT3.TcPOU
FUNCTION_BLOCK FB_StationT3
VAR_IN_OUT
	XpMover			: MC_PlanarMover;
	XpTrack			: ARRAY [*] OF MC_PlanarTrack;
END_VAR
VAR_INPUT
	execute			: BOOL;
END_VAR
VAR_OUTPUT
	bOccupied		: BOOL;
	bBeforeRotate	: BOOL;
	bReady			: BOOL;
END_VAR
VAR
	nState			: INT;
	fbMoveTrack		: FB_XpMoveTrack;
	fbMoveC			: FB_XpMoveC;
	nTargetTrack	: INT;
	bMove			: BOOL;
	bMoveC			: BOOL;
	nRotatePos		: LREAL :=0;
END_VAR

CASE nState OF
	0: //init
	IF execute THEN
		bOccupied := TRUE;//Stationの状態をOccupiedにする
		bReady := FALSE;
		nState := 20;
	END_IF	
	
	20://移動
	bMove:= TRUE;
	nTargetTrack:= E_TrackName.T2_2_ToRotate;
	fbMoveTrack.execute := TRUE;
	
	IF fbMoveTrack.done THEN
		fbMoveTrack.execute:= FALSE;
		bOccupied := FALSE;
		bReady := TRUE;//Stationの状態をReadyにする
		bBeforeRotate := TRUE;//Rotate前の位置まで移動したことをT2に伝える
		bMove:= FALSE;
		nState := 30;
	END_IF
	
	30://回転
	bMoveC := TRUE;
	fbMoveC.execute:= TRUE;
	
	IF fbMoveC.done THEN
		fbMoveC.execute := FALSE;
		bBeforeRotate := FALSE;
		bMoveC:= FALSE;
		nState := 40;
	END_IF
	
	40://T1まで移動
	nTargetTrack:= E_TrackName.T1_1_ToRotate;
	fbMoveTrack.execute:= TRUE;
		nState := 100;
	
	100://initへ戻る
	fbMoveTrack.execute := FALSE;//移動指令を落とす
	nState := 0;
END_CASE

IF bMove THEN
	fbMoveTrack(XpMover:= XpMover, 
				XpTrack:= XpTrack[nTargetTrack]);
ELSIF bMoveC THEN	
	fbMoveC(XpMover:= XpMover, 
			position:= nRotatePos + 360);
END_IF

END_FUNCTION_BLOCK

// ---- POUs/FB/FB_StationT4.TcPOU
FUNCTION_BLOCK FB_StationT4
VAR_IN_OUT
	XpMover			: MC_PlanarMover;
	XpTrack			: ARRAY[*] OF MC_PlanarTrack;
END_VAR
VAR_INPUT
	execute			: BOOL;
END_VAR
VAR_OUTPUT
	bOccupied		: BOOL;
	bReady			: BOOL;
END_VAR
VAR
	nState			: INT;
	fbMoveTrack		: FB_XpMoveTrack;
	nTargetTrack	: INT;
	fbMoveC			: FB_XpMoveC;
	bMoveC: BOOL;
	nRotatePos		: LREAL :=0;
END_VAR

CASE nState OF
	0://init
	IF execute THEN
		bOccupied := TRUE;//Stationの状態をOccupiedにする
		bReady := FALSE;
		nState := 10;
	END_IF
	
	10:
	bMoveC := TRUE;
	fbMoveC.execute := TRUE;
	
	IF fbMoveC.done THEN
		fbMoveC.execute := FALSE;
		bMoveC := FALSE;
		nState := 420;
	END_IF
	
	20://T1まで移動
	ntargetTrack :=E_TrackName.T1_1_ToRotate;
	fbMoveTrack.execute:= TRUE;
		nState := 100;
	
	100://initへ戻る
	fbMoveTrack.execute := FALSE;//移動指令を落とす
	nState := 0;
	
END_CASE

IF bMoveC THEN
	fbMoveTrack(XpMover:= XpMover, 
				XpTrack:= XpTrack[nTargetTrack]);
	fbMoveC(XpMover:= XpMover, 
			position:= nRotatePos + 360);
END_IF

END_FUNCTION_BLOCK

// ---- POUs/FindMoverInArea.TcPOU
FUNCTION FindMoverInArea : INT
VAR_INPUT
	stParam		: ST_StationParams;
END_VAR
VAR_IN_OUT
	XpMover		: ARRAY[*] OF MC_PlanarMover;
END_VAR
VAR
	i 			: DINT;
END_VAR

//初期値0
FindMoverInArea := 0;

//各Moverが指定範囲にいるかサーチする
FOR i:=LOWER_BOUND(XpMover, 1) TO UPPER_BOUND(XpMover ,1) DO
	IF 
	XpMover[i].MCTOPLC.SET.SetPos.x >= stParam.fMinX AND
	XpMover[i].MCTOPLC.SET.SetPos.x <= stParam.fMaxX AND
	XpMover[i].MCTOPLC.SET.SetPos.y >= stParam.fMinY AND
	XpMover[i].MCTOPLC.SET.SetPos.y <= stParam.fMaxY THEN
	//指定範囲にいるMoverの番号を取得
		FindMoverInArea := DINT_TO_INT(i);
		RETURN;
	END_IF
END_FOR

END_FUNCTION

// ---- POUs/FB/FB_XpExternalSetPoint.TcPOU
FUNCTION_BLOCK FB_XpExternalSetPoint
VAR_IN_OUT
	XpMover							: MC_PlanarMover;
	McArrayAxis						: ARRAY [1..6] OF AXIS_REF;
END_VAR
VAR_INPUT
	enable							: BOOL;
	modeExteanlSetPoint				: MC_EXTERNAL_SET_POSITION_MODE;
END_VAR
VAR_OUTPUT
	valid							: BOOL;
	busy							: BOOL;
	error							: BOOL;
	aborted							: BOOL;
END_VAR
VAR
	_XpFeedback						: ARRAY [0.._MAX_XPLANAR_FEEDBACK] OF MC_PlanarFeedback;
END_VAR
VAR
	_sequence						: UINT;
	_i								: UINT;
	_countError						: UINT;
	_SetPosition					: MoverVector;
	_SetVelocity					: MoverVector;
	_SetAcceleration				: MoverVector;
	_OptionsExternalSetPosition		: ST_ExternalSetpointGenerationOptions;
END_VAR
VAR CONSTANT
	_MAX_XPLANAR_FEEDBACK			: UINT := 1;
	_MAX_COUNT_ERROR				: UINT := 5;
	
	_INIT							: UINT := 0000;
	_READY							: UINT := 0001;
	_START_EXTERNAL_SET_POSITION	: UINT := 0011;
	_CHECK_START_EXTERNAL_SET_POSITION	: UINT := 0012;
	_SET_POSITION					: UINT := 0013;
	_STOP_EXTERNAL_SET_POINT		: UINT := 0014;
	_CHECK_STOP_EXTERNAL_SET_POINT	: UINT := 0015;
	_DONE							: UINT := 1000;
	_ERROR							: UINT := 2000;
	_ABORTED						: UINT := 3000;
END_VAR

updateXPlanarFB();
updateReadStatus();
CASE _sequence OF
	_INIT:
		_sequence := _READY;

	_READY:
		IF enable THEN 
			_sequence := _START_EXTERNAL_SET_POSITION; 
			busy := TRUE;
			error := FALSE;
		END_IF

	_START_EXTERNAL_SET_POSITION:
		_OptionsExternalSetPosition.mode := modeExteanlSetPoint;
		XpMover.StartExternalSetpointGeneration(commandFeedback:= _XpFeedback[0], options:= _OptionsExternalSetPosition);
		_sequence := _CHECK_START_EXTERNAL_SET_POSITION;
	
	_CHECK_START_EXTERNAL_SET_POSITION:
		IF _XpFeedback[0].Done THEN _sequence := _SET_POSITION; END_IF
	
	_SET_POSITION:
		valid := TRUE;
		_SetPosition.x := McArrayAxis[1].NcToPlc.ActPos;
		_SetPosition.y := McArrayAxis[2].NcToPlc.ActPos;
		_SetPosition.z := McArrayAxis[3].NcToPlc.ActPos;
		_SetPosition.a := McArrayAxis[4].NcToPlc.ActPos;
		_SetPosition.b := McArrayAxis[5].NcToPlc.ActPos;
		_SetPosition.c := McArrayAxis[6].NcToPlc.ActPos;
		
		_SetVelocity.x := McArrayAxis[1].NcToPlc.ActVelo;
		_SetVelocity.y := McArrayAxis[2].NcToPlc.ActVelo;
		_SetVelocity.z := McArrayAxis[3].NcToPlc.ActVelo;
		_SetVelocity.a := McArrayAxis[4].NcToPlc.ActVelo;
		_SetVelocity.b := McArrayAxis[5].NcToPlc.ActVelo;
		_SetVelocity.c := McArrayAxis[6].NcToPlc.ActVelo;
		
		_SetAcceleration.x := McArrayAxis[1].NcToPlc.ActAcc;
		_SetAcceleration.y := McArrayAxis[2].NcToPlc.ActAcc;
		_SetAcceleration.z := McArrayAxis[3].NcToPlc.ActAcc;
		_SetAcceleration.a := McArrayAxis[4].NcToPlc.ActAcc;
		_SetAcceleration.b := McArrayAxis[5].NcToPlc.ActAcc;
		_SetAcceleration.c := McArrayAxis[6].NcToPlc.ActAcc;
		
		XpMover.SetExternalSetpoint(
			setPosition:= _SetPosition, 
			setVelocity:= _SetVelocity, 
			setAcceleration:= _SetAcceleration);
		
		IF NOT enable THEN
			_sequence := _STOP_EXTERNAL_SET_POINT;
		END_IF
	
	_STOP_EXTERNAL_SET_POINT:
		XpMover.StopExternalSetpointGeneration(commandFeedback:= _XpFeedback[1]);
		_sequence := _CHECK_STOP_EXTERNAL_SET_POINT;
	
	_CHECK_STOP_EXTERNAL_SET_POINT:
		IF _XpFeedback[1].Done THEN _sequence := _DONE; END_IF
		
	_DONE:
		valid := FALSE;
		busy := FALSE;
		_sequence := _READY;
		
	_ERROR:
		valid := FALSE;
		busy := FALSE;
		error := TRUE;
		_sequence := _READY;
END_CASE

ACTION updateReadStatus:
FOR _i:=1 TO 6 DO
	McArrayAxis[_i].ReadStatus();
END_FOR
END_ACTION

ACTION updateXPlanarFB:
FOR _i:=0 TO _MAX_XPLANAR_FEEDBACK DO
	_XpFeedback[_i].Update();
END_FOR
END_ACTION

END_FUNCTION_BLOCK

// ---- POUs/FB/FB_XpLeaveTrack.TcPOU
FUNCTION_BLOCK FB_XpLeaveTrack
VAR_IN_OUT
	XpMover							: MC_PlanarMover;
	XpTrack							: MC_PlanarTrack;
END_VAR
VAR_INPUT
	execute							: BOOL;
END_VAR
VAR_OUTPUT
	done							: BOOL;
	busy							: BOOL;
	error							: BOOL;
	aborted							: BOOL;
END_VAR
VAR
	_XpFeedback						: ARRAY [0.._MAX_XPLANAR_FEEDBACK] OF MC_PlanarFeedback;
	_XpTargetPosition 				: PositionXYC;
	_XpCondition		 			: DynamicConstraint_PathXY;
END_VAR
VAR
	_sequence						: UINT;
	_i								: UINT;
	_countError						: UINT;
END_VAR
VAR CONSTANT
	_MAX_XPLANAR_FEEDBACK			: UINT := 1;
	_MAX_COUNT_ERROR				: UINT := 5;
	
	_INIT							: UINT := 0000;
	_READY							: UINT := 0001;
	_LEAVE_TRACK					: UINT := 0011;
	_CHECK_LEAVE_TRACK				: UINT := 0012;
	_DONE							: UINT := 1000;
	_ERROR							: UINT := 2000;
	_ABORTED						: UINT := 3000;
END_VAR

updateXPlanarFB();
CASE _sequence OF
	_INIT:
		_sequence := _READY;
		
	_READY:
		IF execute THEN
			busy := TRUE;
			_sequence := _LEAVE_TRACK;
			setInputVariables();
		END_IF
		
	_LEAVE_TRACK:
		_XpCondition.SetValuesVADJ(
			V:= 100, 
			A:= 2000, 
			D:= 2000, 
			J:= 20000);
		_XpTargetPosition.SetValuesXYC(
			x:= XpMover.MCTOPLC.ACT.ActPos.x, 
			y:= XpMover.MCTOPLC.ACT.ActPos.y, 
			c:= XpMover.MCTOPLC.ACT.ActPos.c);
		XpMover.LeaveTrack(commandFeedback:= _XpFeedback[0], 
			targetPosition:= _XpTargetPosition, 
			constraint:= _XpCondition, 
			options:= 0);
		_sequence := _CHECK_LEAVE_TRACK;
		
	_CHECK_LEAVE_TRACK:
		IF _XpFeedback[0].Done THEN
			_countError := 0;
			_sequence := _DONE;
		ELSIF _XpFeedback[0].Error THEN
			_countError := _countError + 1;
			_sequence := _LEAVE_TRACK;
		ELSIF _XpFeedback[0].Aborted THEN
			_countError := 0;
			_sequence := _ABORTED;
		END_IF
		IF _countError > _MAX_COUNT_ERROR THEN
			_countError := 0;
			_sequence := _ERROR;
		END_IF
		
	_DONE:
		done := TRUE;
		busy := FALSE;
		IF NOT execute THEN
			done := FALSE;
			_sequence := _READY;
		END_IF
	
	_ERROR:
		error := TRUE;
		busy := FALSE;
		IF NOT execute THEN
			error := FALSE;
			_sequence := _READY;
		END_IF
		
	_ABORTED:
		aborted := TRUE;
		busy := FALSE;
		IF NOT execute THEN
			aborted := FALSE;
			_sequence := _READY;
		END_IF
END_CASE

ACTION setInputVariables:

END_ACTION

ACTION updateXPlanarFB:
FOR _i:=0 TO _MAX_XPLANAR_FEEDBACK DO
	_XpFeedback[_i].Update();
END_FOR
END_ACTION

END_FUNCTION_BLOCK

// ---- POUs/FB/FB_XpMoveA.TcPOU
FUNCTION_BLOCK FB_XpMoveA
VAR_IN_OUT
	XpMover							: MC_PlanarMover;
END_VAR
VAR_INPUT
	execute							: BOOL;
	position						: LREAL := 2;
	velocity						: LREAL := 100;
	acceleration					: LREAL := 2000;
	jerk							: LREAL := 20000;
END_VAR
VAR_OUTPUT
	done							: BOOL;
	busy							: BOOL;
	error							: BOOL;
	aborted							: BOOL;
END_VAR
VAR
	_XpFeedback						: ARRAY [0.._MAX_XPLANAR_FEEDBACK] OF MC_PlanarFeedback;
	_XpCondition		 			: DynamicConstraint_Coordinates;
END_VAR
VAR
	_sequence						: UINT;
	_i								: UINT;
	_countError						: UINT;
	_position						: LREAL;
	_velocity						: LREAL;
	_acceleration					: LREAL;
	_jerk							: LREAL;
END_VAR
VAR CONSTANT
	_MAX_XPLANAR_FEEDBACK			: UINT := 1;
	_MAX_COUNT_ERROR				: UINT := 5;
	
	_INIT							: UINT := 0000;
	_READY							: UINT := 0001;
	_MOVE_A							: UINT := 0011;
	_CHECK_MOVE_A					: UINT := 0012;
	_DONE							: UINT := 1000;
	_ERROR							: UINT := 2000;
	_ABORTED						: UINT := 3000;
END_VAR

updateXPlanarFB();
CASE _sequence OF
	_INIT:
		_XpCondition.AddLimit(
			Coordinate:= Coord_Mcs_A1, 
			V:= velocity, 
			A:= acceleration, 
			D:= acceleration, 
			J:= jerk);
		_sequence := _READY;
	
	_READY:
		IF execute THEN
			busy := TRUE;
			_sequence := _MOVE_A;
			setInputVariables();
		END_IF
		
	_MOVE_A:
		_XpCondition.SetLimit(
			Coordinate:= Coord_Mcs_A1, 
			V:= _velocity, 
			A:= _acceleration, 
			D:= _acceleration, 
			J:= _jerk);
		XpMover.MoveA(commandFeedback:= _XpFeedback[0], 
			targetPosition:= _position, 
			constraint:= _XpCondition);
		_sequence := _CHECK_MOVE_A;
		
	_CHECK_MOVE_A:
		IF _XpFeedback[0].Done THEN
			_countError := 0;
			_sequence := _DONE;
		ELSIF _XpFeedback[0].Error THEN
			_countError := _countError + 1;
			_sequence := _MOVE_A;
		END_IF
		IF _countError > _MAX_COUNT_ERROR THEN
			_countError := 0;
			_sequence := _ERROR;
		END_IF
		
	_DONE:
		done := TRUE;
		busy := FALSE;
		IF NOT execute THEN
			done := FALSE;
			_sequence := _READY;
		END_IF
	
	_ERROR:
		error := TRUE;
		busy := FALSE;
		IF NOT execute THEN
			error := FALSE;
			_sequence := _READY;
		END_IF
		
	_ABORTED:
		aborted := TRUE;
		busy := FALSE;
		IF NOT execute THEN
			aborted := FALSE;
			_sequence := _READY;
		END_IF
END_CASE

ACTION setInputVariables:
_position := position;
_velocity := velocity;
_acceleration := acceleration;
_jerk := jerk;
END_ACTION

ACTION updateXPlanarFB:
FOR _i:=0 TO _MAX_XPLANAR_FEEDBACK DO
	_XpFeedback[_i].Update();
END_FOR
END_ACTION

END_FUNCTION_BLOCK

// ---- POUs/FB/FB_XpMoveB.TcPOU
FUNCTION_BLOCK FB_XpMoveB
VAR_IN_OUT
	XpMover							: MC_PlanarMover;
END_VAR
VAR_INPUT
	execute							: BOOL;
	position						: LREAL := 2;
	velocity						: LREAL := 100;
	acceleration					: LREAL := 2000;
	jerk							: LREAL := 20000;
END_VAR
VAR_OUTPUT
	done							: BOOL;
	busy							: BOOL;
	error							: BOOL;
	aborted							: BOOL;
END_VAR
VAR
	_XpFeedback						: ARRAY [0.._MAX_XPLANAR_FEEDBACK] OF MC_PlanarFeedback;
	_XpCondition		 			: DynamicConstraint_Coordinates;
END_VAR
VAR
	_sequence						: UINT;
	_i								: UINT;
	_countError						: UINT;
	_position						: LREAL;
	_velocity						: LREAL;
	_acceleration					: LREAL;
	_jerk							: LREAL;
END_VAR
VAR CONSTANT
	_MAX_XPLANAR_FEEDBACK			: UINT := 1;
	_MAX_COUNT_ERROR				: UINT := 5;
	
	_INIT							: UINT := 0000;
	_READY							: UINT := 0001;
	_MOVE_B							: UINT := 0011;
	_CHECK_MOVE_B					: UINT := 0012;
	_DONE							: UINT := 1000;
	_ERROR							: UINT := 2000;
	_ABORTED						: UINT := 3000;
END_VAR

updateXPlanarFB();
CASE _sequence OF
	_INIT:
		_XpCondition.AddLimit(
			Coordinate:= Coord_Mcs_B1, 
			V:= velocity, 
			A:= acceleration, 
			D:= acceleration, 
			J:= jerk);
		_sequence := _READY;
	
	_READY:
		IF execute THEN
			busy := TRUE;
			_sequence := _MOVE_B;
			setInputVariables();
		END_IF
		
	_MOVE_B:
		_XpCondition.SetLimit(
			Coordinate:= Coord_Mcs_B1, 
			V:= _velocity, 
			A:= _acceleration, 
			D:= _acceleration, 
			J:= _jerk);
		XpMover.MoveB(commandFeedback:= _XpFeedback[0], 
			targetPosition:= _position, 
			constraint:= _XpCondition);
		_sequence := _CHECK_MOVE_B;
		
	_CHECK_MOVE_B:
		IF _XpFeedback[0].Done THEN
			_countError := 0;
			_sequence := _DONE;
		ELSIF _XpFeedback[0].Error THEN
			_countError := _countError + 1;
			_sequence := _MOVE_B;
		END_IF
		IF _countError > _MAX_COUNT_ERROR THEN
			_countError := 0;
			_sequence := _ERROR;
		END_IF
		
	_DONE:
		done := TRUE;
		busy := FALSE;
		IF NOT execute THEN
			done := FALSE;
			_sequence := _READY;
		END_IF
	
	_ERROR:
		error := TRUE;
		busy := FALSE;
		IF NOT execute THEN
			error := FALSE;
			_sequence := _READY;
		END_IF
		
	_ABORTED:
		aborted := TRUE;
		busy := FALSE;
		IF NOT execute THEN
			aborted := FALSE;
			_sequence := _READY;
		END_IF
END_CASE

ACTION setInputVariables:
_position := position;
_velocity := velocity;
_acceleration := acceleration;
_jerk := jerk;
END_ACTION

ACTION updateXPlanarFB:
FOR _i:=0 TO _MAX_XPLANAR_FEEDBACK DO
	_XpFeedback[_i].Update();
END_FOR
END_ACTION

END_FUNCTION_BLOCK

// ---- POUs/FB/FB_XpMoveXY.TcPOU
FUNCTION_BLOCK FB_XpMoveXY
VAR_IN_OUT
	XpMover							: MC_PlanarMover;
END_VAR
VAR_INPUT
	execute							: BOOL;
	position_x						: LREAL := 160;
	position_y						: LREAL := 160;	
	velocity						: LREAL := 100;
	acceleration					: LREAL := 2000;
	jerk							: LREAL := 20000;
END_VAR
VAR_OUTPUT
	done							: BOOL;
	busy							: BOOL;
	error							: BOOL;
	aborted							: BOOL;
END_VAR
VAR
	_XpFeedback						: ARRAY [0.._MAX_XPLANAR_FEEDBACK] OF MC_PlanarFeedback;
	_XpTargetPosition 				: PositionXYC;
	_XpCondition		 			: DynamicConstraint_PathXY;
END_VAR
VAR
	_sequence						: UINT;
	_i								: UINT;
	_countError						: UINT;
	_position_x						: LREAL;
	_position_y						: LREAL;
	_velocity						: LREAL;
	_acceleration					: LREAL;
	_jerk							: LREAL;
END_VAR
VAR CONSTANT
	_MAX_XPLANAR_FEEDBACK			: UINT := 1;
	_MAX_COUNT_ERROR				: UINT := 5;
	
	_INIT							: UINT := 0000;
	_READY							: UINT := 0001;
	_MOVE_TO_POSITION				: UINT := 0011;
	_CHECK_MOVE_TO_POSITION			: UINT := 0012;
	_DONE							: UINT := 1000;
	_ERROR							: UINT := 2000;
	_ABORTED						: UINT := 3000;
END_VAR

updateXPlanarFB();
CASE _sequence OF
	_INIT:
		_sequence := _READY;
		
	_READY:
		IF execute THEN
			busy := TRUE;
			_sequence := _MOVE_TO_POSITION;
			setInputVariables();
		END_IF
		
	_MOVE_TO_POSITION:
		_XpCondition.SetValuesVADJ(
			V:= _velocity, 
			A:= _acceleration, 
			D:= _acceleration, 
			J:= _jerk);
		_XpTargetPosition.SetValuesXYC(
			x:= _position_x, 
			y:= _position_y, 
			c:= XpMover.MCTOPLC.ACT.ActPos.c);
		XpMover.MoveToPosition(commandFeedback:= _XpFeedback[0], 
			targetPosition:= _XpTargetPosition, 
			constraint:= _XpCondition, 
			options:= 0);
		_sequence := _CHECK_MOVE_TO_POSITION;
		
	_CHECK_MOVE_TO_POSITION:
		IF _XpFeedback[0].Done THEN
			_countError := 0;
			_sequence := _DONE;
		ELSIF _XpFeedback[0].Error THEN
			_countError := _countError + 1;
			_sequence := _MOVE_TO_POSITION;
		END_IF
		IF _countError > _MAX_COUNT_ERROR THEN
			_countError := 0;
			_sequence := _ERROR;
		END_IF
		
	_DONE:
		done := TRUE;
		busy := FALSE;
		IF NOT execute THEN
			done := FALSE;
			_sequence := _READY;
		END_IF
	
	_ERROR:
		error := TRUE;
		busy := FALSE;
		IF NOT execute THEN
			error := FALSE;
			_sequence := _READY;
		END_IF
		
	_ABORTED:
		aborted := TRUE;
		busy := FALSE;
		IF NOT execute THEN
			aborted := FALSE;
			_sequence := _READY;
		END_IF
END_CASE

ACTION setInputVariables:
_position_x := position_x;
_position_y := position_y;
_velocity := velocity;
_acceleration := acceleration;
_jerk := jerk;
END_ACTION

ACTION updateXPlanarFB:
FOR _i:=0 TO _MAX_XPLANAR_FEEDBACK DO
	_XpFeedback[_i].Update();
END_FOR
END_ACTION

END_FUNCTION_BLOCK

// ---- POUs/FB/FB_XpMoveZ.TcPOU
FUNCTION_BLOCK FB_XpMoveZ
VAR_IN_OUT
	XpMover							: MC_PlanarMover;
END_VAR
VAR_INPUT
	execute							: BOOL;
	position						: LREAL := 2;
	velocity						: LREAL := 100;
	acceleration					: LREAL := 2000;
	jerk							: LREAL := 20000;
END_VAR
VAR_OUTPUT
	done							: BOOL;
	busy							: BOOL;
	error							: BOOL;
	aborted							: BOOL;
END_VAR
VAR
	_XpFeedback						: ARRAY [0.._MAX_XPLANAR_FEEDBACK] OF MC_PlanarFeedback;
	_XpCondition		 			: DynamicConstraint_Coordinates;
END_VAR
VAR
	_sequence						: UINT;
	_i								: UINT;
	_countError						: UINT;
	_position						: LREAL;
	_velocity						: LREAL;
	_acceleration					: LREAL;
	_jerk							: LREAL;
END_VAR
VAR CONSTANT
	_MAX_XPLANAR_FEEDBACK			: UINT := 1;
	_MAX_COUNT_ERROR				: UINT := 5;
	
	_INIT							: UINT := 0000;
	_READY							: UINT := 0001;
	_MOVE_Z							: UINT := 0011;
	_CHECK_MOVE_Z					: UINT := 0012;
	_DONE							: UINT := 1000;
	_ERROR							: UINT := 2000;
	_ABORTED						: UINT := 3000;
END_VAR

updateXPlanarFB();
CASE _sequence OF
	_INIT:
		_XpCondition.AddLimit(
			Coordinate:= Coord_Mcs_Z, 
			V:= velocity, 
			A:= acceleration, 
			D:= acceleration, 
			J:= jerk);
		_sequence := _READY;
	
	_READY:
		IF execute THEN
			busy := TRUE;
			_sequence := _MOVE_Z;
			setInputVariables();
		END_IF
		
	_MOVE_Z:
		_XpCondition.SetLimit(
			Coordinate:= Coord_Mcs_Z, 
			V:= _velocity, 
			A:= _acceleration, 
			D:= _acceleration, 
			J:= _jerk);
		XpMover.MoveZ(commandFeedback:= _XpFeedback[0], 
			targetPosition:= _position, 
			constraint:= _XpCondition);
		_sequence := _CHECK_MOVE_Z;
		
	_CHECK_MOVE_Z:
		IF _XpFeedback[0].Done THEN
			_countError := 0;
			_sequence := _DONE;
		ELSIF _XpFeedback[0].Error THEN
			_countError := _countError + 1;
			_sequence := _MOVE_Z;
		END_IF
		IF _countError > _MAX_COUNT_ERROR THEN
			_countError := 0;
			_sequence := _ERROR;
		END_IF
		
	_DONE:
		done := TRUE;
		busy := FALSE;
		IF NOT execute THEN
			done := FALSE;
			_sequence := _READY;
		END_IF
	
	_ERROR:
		error := TRUE;
		busy := FALSE;
		IF NOT execute THEN
			error := FALSE;
			_sequence := _READY;
		END_IF
		
	_ABORTED:
		aborted := TRUE;
		busy := FALSE;
		IF NOT execute THEN
			aborted := FALSE;
			_sequence := _READY;
		END_IF
END_CASE

ACTION setInputVariables:
_position := position;
_velocity := velocity;
_acceleration := acceleration;
_jerk := jerk;
END_ACTION

ACTION updateXPlanarFB:
FOR _i:=0 TO _MAX_XPLANAR_FEEDBACK DO
	_XpFeedback[_i].Update();
END_FOR
END_ACTION

END_FUNCTION_BLOCK

// ---- POUs/FB/FB_XpParallel.TcPOU
FUNCTION_BLOCK FB_XpParallel
VAR_INPUT
END_VAR
VAR_OUTPUT
END_VAR
VAR
END_VAR

END_FUNCTION_BLOCK

// ---- POUs/FB/FB_XpReset.TcPOU
FUNCTION_BLOCK FB_XpReset
VAR_IN_OUT
	XpMover							: MC_PlanarMover;
END_VAR
VAR_INPUT
	execute							: BOOL;
END_VAR
VAR_OUTPUT
	done							: BOOL;
	busy							: BOOL;
	error							: BOOL;
	aborted							: BOOL;
END_VAR
VAR
	_XpFeedback						: ARRAY [0.._MAX_XPLANAR_FEEDBACK] OF MC_PlanarFeedback;
	_XpCondition		 			: DynamicConstraint_Coordinates;
END_VAR
VAR
	_sequence						: UINT;
	_i								: UINT;
	_countError						: UINT;
END_VAR
VAR CONSTANT
	_MAX_XPLANAR_FEEDBACK			: UINT := 1;
	_MAX_COUNT_ERROR				: UINT := 5;
	
	_INIT							: UINT := 0000;
	_READY							: UINT := 0001;
	_RESET							: UINT := 0011;
	_CHECK_RESET					: UINT := 0012;
	_DONE							: UINT := 1000;
	_ERROR							: UINT := 2000;
	_ABORTED						: UINT := 3000;
END_VAR

updateXPlanarFB();
CASE _sequence OF
	_INIT:
		_sequence := _READY;
	
	_READY:
		IF execute THEN
			busy := TRUE;
			_sequence := _RESET;
			setInputVariables();
		END_IF
		
	_RESET:
		XpMover.Reset(commandFeedback:= _XpFeedback[0]);
		_sequence := _CHECK_RESET;
		
	_CHECK_RESET:
		IF _XpFeedback[0].Done THEN
			_countError := 0;
			_sequence := _DONE;
		ELSIF _XpFeedback[0].Error THEN
			_countError := _countError + 1;
			_sequence := _RESET;
		END_IF
		IF _countError > _MAX_COUNT_ERROR THEN
			_countError := 0;
			_sequence := _ERROR;
		END_IF
		
	_DONE:
		done := TRUE;
		busy := FALSE;
		IF NOT execute THEN
			done := FALSE;
			_sequence := _READY;
		END_IF
	
	_ERROR:
		error := TRUE;
		busy := FALSE;
		IF NOT execute THEN
			error := FALSE;
			_sequence := _READY;
		END_IF
		
	_ABORTED:
		aborted := TRUE;
		busy := FALSE;
		IF NOT execute THEN
			aborted := FALSE;
			_sequence := _READY;
		END_IF
END_CASE

ACTION setInputVariables:
_position := position;
_velocity := velocity;
_acceleration := acceleration;
_jerk := jerk;
END_ACTION

ACTION updateXPlanarFB:
FOR _i:=0 TO _MAX_XPLANAR_FEEDBACK DO
	_XpFeedback[_i].Update();
END_FOR
END_ACTION

END_FUNCTION_BLOCK

// ---- GlobalTextList.TcGTLO
TEXTLIST GlobalTextList
  748 = '%d'
  410 = 'C'
  834 = 'C_Rotetion'
  624 = 'C_Rotetion Value'
  785 = 'Disable'
  196 = 'Enable'
  18 = 'mm/s'
  557 = 'MoveC(Rotation)'
  220 = 'Mover No.'
  270 = 'Mover1'
  972 = 'Mover2'
  915 = 'Mover3'
  52 = 'MoveXY'
  945 = 'Point To Move'
  667 = 'realtime position'
  82 = 'Realtime Position'
  318 = 'Reset'
  960 = 'RESET'
  796 = 'Restart'
  740 = 'Start'
  131 = 'Stop'
  567 = 'X'
  477 = 'Y'
  653 = '衝突'
  387 = '衝突回避'
  347 = '衝突回避\nError'
  291 = '衝突回避Error'
  968 = '運転準備'
  378 = '運転開始'
END_TEXTLIST

// ---- VISUs/Visualization.TcVIS
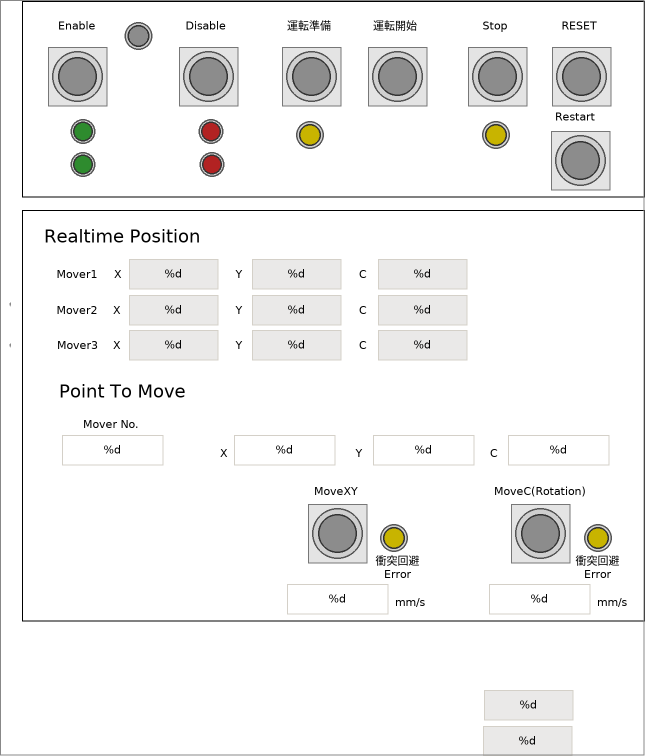
VISUALIZATION Visualization  // 645x756
    RoundedRectangle (22,1 623x196)
    RoundedRectangle (22,210 623x411)
    RockerSwitch (10,302 0x4), behaviour: TOGGLE, style: Switch-RockerSwitch-Gray
    PushSwitch (46,47 63x59), variable: MAIN.exeXpEnableMover, behaviour: TOGGLE, style: Switch-PushSwitch-Gray
    PushSwitch (177,47 63x59), variable: MAIN.exeXpDisableMover, behaviour: TOGGLE, style: Switch-PushSwitch-Gray
    Label (43,15 68x22), "Enable"
    Label (172,15 68x22), "Disable"
    Label (275,15 68x22), "運転準備"
    Label (541,106 68x22), "Restart"
    PushSwitch (280,47 63x59), variable: MAIN.exePreStartPB, behaviour: TOGGLE, style: Switch-PushSwitch-Gray
    PushSwitch (549,131 63x59), variable: MAIN.exerestartPB, behaviour: TOGGLE, style: Switch-PushSwitch-Gray
    PushSwitch (306,504 63x59), variable: MAIN.exeMoveXY, behaviour: TOGGLE, style: Switch-PushSwitch-Gray
    Textfield (234,435 101x30), "%d", text variable: MAIN.nManualX
        OnMouseClick: write the text variable via Default
    Textfield (373,435 101x30), "%d", text variable: MAIN.nManualY
        OnMouseClick: write the text variable via Default
    Textfield (508,435 101x30), "%d", text variable: MAIN.nManualC
        OnMouseClick: write the text variable via Default
    Label (168,442 112x23), "X"
    Label (303,442 112x23), "Y"
    Label (438,442 112x23), "C"
    Label (280,480 112x23), "MoveXY"
    Label (484,480 112x23), "MoveC(Rotation)"
    PushSwitch (509,504 63x59), variable: MAIN.exeMoveC, behaviour: TOGGLE, style: Switch-PushSwitch-Gray
    Textfield (62,435 101x30), "%d", text variable: MAIN.nMover
        OnMouseClick: write the text variable via Default
    Label (55,413 112x23), "Mover No."
    Lamp1 (378,519 32x38), variable: MAIN.ManualCollisionError[0], style: Lamp-Lamp1-Yellow
    Lamp1 (582,519 32x38), variable: MAIN.ManualCollisionError[1], style: Lamp-Lamp1-Yellow
    Lamp1 (294,116 32x38), variable: MAIN.bJoinDone, style: Lamp-Lamp1-Yellow
    Label (367,548 61x39), "衝突回避 Error"
    Label (567,548 61x39), "衝突回避 Error"
    Lamp1 (62,117 42x29), variable: MAIN.bMoverEnable[1], style: Lamp-Lamp1-Green
    Lamp1 (62,150 42x29), variable: MAIN.bMoverEnable[2], style: Lamp-Lamp1-Green
    Lamp1 (191,150 42x29), variable: MAIN.bMoverDisable[2], style: Lamp-Lamp1-Red
    Lamp1 (190,117 42x29), variable: MAIN.bMoverDisable[1], style: Lamp-Lamp1-Red
    PushSwitch (466,47 63x59), variable: MAIN.exeStop_os, behaviour: TOGGLE, style: Switch-PushSwitch-Gray
    Label (461,15 68x22), "Stop"
    Textfield (129,259 89x30), "%d", text variable: MAIN.VisVar[1][0]
    Textfield (252,259 89x30), "%d", text variable: MAIN.VisVar[1][1]
    Textfield (484,690 89x30), "%d", text variable: MAIN.VisVar[1][2]
    Label (62,263 112x23), "X"
    Label (183,263 112x23), "Y"
    Label (307,263 112x23), "C"
    Label (61,299 112x23), "X"
    Textfield (252,295 89x30), "%d", text variable: MAIN.VisVar[2][1]
    Textfield (483,726 89x30), "%d", text variable: MAIN.VisVar[2][2]
    Label (183,299 112x23), "Y"
    Label (307,299 112x23), "C"
    Textfield (129,295 89x30), "%d", text variable: MAIN.VisVar[2][0]
    Label (36,225 173x23), "Realtime Position"
    Label (21,263 112x23), "Mover1"
    Label (21,299 112x23), "Mover2"
    Label (36,380 173x23), "Point To Move"
    Textfield (489,584 101x30), "%d", text variable: MAIN.ValueC
        OnMouseClick: write the text variable via Default
    Label (545,15 68x22), "RESET"
    PushSwitch (550,47 63x59), variable: MAIN.exeresetPB, behaviour: TOGGLE, style: Switch-PushSwitch-Gray
    Textfield (378,259 89x30), "%d", text variable: MAIN.VisVar[1][3]
    Textfield (378,295 89x30), "%d", text variable: MAIN.VisVar[2][2]
    Textfield (287,584 101x30), "%d", text variable: MAIN.valueV
        OnMouseClick: write the text variable via Default
    Label (385,591 50x23), "mm/s"
    Label (587,591 50x23), "mm/s"
    Lamp1 (480,116 32x38), variable: MAIN.exeStop, style: Lamp-Lamp1-Yellow
    Lamp1 (121,20 35x32), variable: MAIN.fbAutoScan.bDone, style: Lamp-Lamp1-Gray
    RockerSwitch (10,343 0x4), behaviour: TOGGLE, style: Switch-RockerSwitch-Gray
    Label (61,334 112x23), "X"
    Label (183,334 112x23), "Y"
    Label (307,334 112x23), "C"
    Label (36,334 83x23), "Mover3"
    Textfield (129,330 89x30), "%d", text variable: MAIN.VisVar[3][0]
    Textfield (252,330 89x30), "%d", text variable: MAIN.VisVar[3][1]
    Textfield (378,330 89x30), "%d", text variable: MAIN.VisVar[3][2]
    Label (361,15 68x22), "運転開始"
    PushSwitch (366,47 63x59), variable: MAIN.exeStartPB, behaviour: TOGGLE, style: Switch-PushSwitch-Gray
END_VISUALIZATION
